{attribute addProperty BoxType "IODEVICETYPE_ETHERCATPROT"}
{attribute addProperty Id "DevCtrlAT %Q*UINT1620Frm0CtrlAT %Q*UINT1620Frm0WcCtrlAT %Q*UINT1620Frm1CtrlAT %Q*UINT1620Frm1WcCtrlAT %Q*UINT1620Frm2CtrlAT %Q*UINT1620Frm2WcCtrlAT %Q*UINT1620Frm3CtrlAT %Q*UINT1620Frm3WcCtrlAT %Q*UINT1620Frm4CtrlAT %Q*UINT1620Frm4WcCtrlAT %Q*UINT1620Frm5CtrlAT %Q*UINT1620Frm5WcCtrlAT %Q*UINT1620Frm6CtrlAT %Q*UINT1620Frm6WcCtrlAT %Q*UINT1620Frm7CtrlAT %Q*UINT1620Frm7WcCtrlAT %Q*UINT1620Frm8CtrlAT %Q*UINT1620Frm8WcCtrlAT %Q*UINT1620Frm9CtrlAT %Q*UINT1620Frm9WcCtrlAT %Q*UINT1620Frm10CtrlAT %Q*UINT1620Frm10WcCtrlAT %Q*UINT1620Frm11CtrlAT %Q*UINT1620Frm11WcCtrlAT %Q*UINT1620Frm12CtrlAT %Q*UINT1620Frm12WcCtrlAT %Q*UINT1620Frm13CtrlAT %Q*UINT1620Frm13WcCtrlAT %Q*UINT1620Frm14CtrlAT %Q*UINT1620Frm14WcCtrlAT %Q*UINT1620Frm15CtrlAT %Q*UINT1620Frm15WcCtrlAT %Q*UINT1620Frm16CtrlAT %Q*UINT1620Frm16WcCtrlAT %Q*UINT1620Frm17CtrlAT %Q*UINT1620Frm17WcCtrlAT %Q*UINT1620Frm18CtrlAT %Q*UINT1620Frm18WcCtrlAT %Q*UINT1620Frm19CtrlAT %Q*UINT1620Frm19WcCtrlAT %Q*UINT1620Frm20CtrlAT %Q*UINT1620Frm20WcCtrlAT %Q*UINT1620Frm21CtrlAT %Q*UINT1620Frm21WcCtrlAT %Q*UINT1620Frm22CtrlAT %Q*UINT1620Frm22WcCtrlAT %Q*UINT1620Frm23CtrlAT %Q*UINT1620Frm23WcCtrlAT %Q*UINT1620Frm24CtrlAT %Q*UINT1620Frm24WcCtrlAT %Q*UINT1620Frm25CtrlAT %Q*UINT1620Frm25WcCtrlAT %Q*UINT1620"}
{attribute addProperty CRC "1204938755"}
{attribute addProperty SizeInBites "848"}
{attribute addProperty SizeInBytes "106"}
TYPE Outputs_47D1E803 :
STRUCT
	{attribute addProperty Name "DevCtrl"}
	DevCtrl AT %Q* : UINT;
	{attribute addProperty Name "Frm0Ctrl"}
	Frm0Ctrl AT %Q* : UINT;
	{attribute addProperty Name "Frm0WcCtrl"}
	Frm0WcCtrl AT %Q* : UINT;
	{attribute addProperty Name "Frm1Ctrl"}
	Frm1Ctrl AT %Q* : UINT;
	{attribute addProperty Name "Frm1WcCtrl"}
	Frm1WcCtrl AT %Q* : UINT;
	{attribute addProperty Name "Frm2Ctrl"}
	Frm2Ctrl AT %Q* : UINT;
	{attribute addProperty Name "Frm2WcCtrl"}
	Frm2WcCtrl AT %Q* : UINT;
	{attribute addProperty Name "Frm3Ctrl"}
	Frm3Ctrl AT %Q* : UINT;
	{attribute addProperty Name "Frm3WcCtrl"}
	Frm3WcCtrl AT %Q* : UINT;
	{attribute addProperty Name "Frm4Ctrl"}
	Frm4Ctrl AT %Q* : UINT;
	{attribute addProperty Name "Frm4WcCtrl"}
	Frm4WcCtrl AT %Q* : UINT;
	{attribute addProperty Name "Frm5Ctrl"}
	Frm5Ctrl AT %Q* : UINT;
	{attribute addProperty Name "Frm5WcCtrl"}
	Frm5WcCtrl AT %Q* : UINT;
	{attribute addProperty Name "Frm6Ctrl"}
	Frm6Ctrl AT %Q* : UINT;
	{attribute addProperty Name "Frm6WcCtrl"}
	Frm6WcCtrl AT %Q* : UINT;
	{attribute addProperty Name "Frm7Ctrl"}
	Frm7Ctrl AT %Q* : UINT;
	{attribute addProperty Name "Frm7WcCtrl"}
	Frm7WcCtrl AT %Q* : UINT;
	{attribute addProperty Name "Frm8Ctrl"}
	Frm8Ctrl AT %Q* : UINT;
	{attribute addProperty Name "Frm8WcCtrl"}
	Frm8WcCtrl AT %Q* : UINT;
	{attribute addProperty Name "Frm9Ctrl"}
	Frm9Ctrl AT %Q* : UINT;
	{attribute addProperty Name "Frm9WcCtrl"}
	Frm9WcCtrl AT %Q* : UINT;
	{attribute addProperty Name "Frm10Ctrl"}
	Frm10Ctrl AT %Q* : UINT;
	{attribute addProperty Name "Frm10WcCtrl"}
	Frm10WcCtrl AT %Q* : UINT;
	{attribute addProperty Name "Frm11Ctrl"}
	Frm11Ctrl AT %Q* : UINT;
	{attribute addProperty Name "Frm11WcCtrl"}
	Frm11WcCtrl AT %Q* : UINT;
	{attribute addProperty Name "Frm12Ctrl"}
	Frm12Ctrl AT %Q* : UINT;
	{attribute addProperty Name "Frm12WcCtrl"}
	Frm12WcCtrl AT %Q* : UINT;
	{attribute addProperty Name "Frm13Ctrl"}
	Frm13Ctrl AT %Q* : UINT;
	{attribute addProperty Name "Frm13WcCtrl"}
	Frm13WcCtrl AT %Q* : UINT;
	{attribute addProperty Name "Frm14Ctrl"}
	Frm14Ctrl AT %Q* : UINT;
	{attribute addProperty Name "Frm14WcCtrl"}
	Frm14WcCtrl AT %Q* : UINT;
	{attribute addProperty Name "Frm15Ctrl"}
	Frm15Ctrl AT %Q* : UINT;
	{attribute addProperty Name "Frm15WcCtrl"}
	Frm15WcCtrl AT %Q* : UINT;
	{attribute addProperty Name "Frm16Ctrl"}
	Frm16Ctrl AT %Q* : UINT;
	{attribute addProperty Name "Frm16WcCtrl"}
	Frm16WcCtrl AT %Q* : UINT;
	{attribute addProperty Name "Frm17Ctrl"}
	Frm17Ctrl AT %Q* : UINT;
	{attribute addProperty Name "Frm17WcCtrl"}
	Frm17WcCtrl AT %Q* : UINT;
	{attribute addProperty Name "Frm18Ctrl"}
	Frm18Ctrl AT %Q* : UINT;
	{attribute addProperty Name "Frm18WcCtrl"}
	Frm18WcCtrl AT %Q* : UINT;
	{attribute addProperty Name "Frm19Ctrl"}
	Frm19Ctrl AT %Q* : UINT;
	{attribute addProperty Name "Frm19WcCtrl"}
	Frm19WcCtrl AT %Q* : UINT;
	{attribute addProperty Name "Frm20Ctrl"}
	Frm20Ctrl AT %Q* : UINT;
	{attribute addProperty Name "Frm20WcCtrl"}
	Frm20WcCtrl AT %Q* : UINT;
	{attribute addProperty Name "Frm21Ctrl"}
	Frm21Ctrl AT %Q* : UINT;
	{attribute addProperty Name "Frm21WcCtrl"}
	Frm21WcCtrl AT %Q* : UINT;
	{attribute addProperty Name "Frm22Ctrl"}
	Frm22Ctrl AT %Q* : UINT;
	{attribute addProperty Name "Frm22WcCtrl"}
	Frm22WcCtrl AT %Q* : UINT;
	{attribute addProperty Name "Frm23Ctrl"}
	Frm23Ctrl AT %Q* : UINT;
	{attribute addProperty Name "Frm23WcCtrl"}
	Frm23WcCtrl AT %Q* : UINT;
	{attribute addProperty Name "Frm24Ctrl"}
	Frm24Ctrl AT %Q* : UINT;
	{attribute addProperty Name "Frm24WcCtrl"}
	Frm24WcCtrl AT %Q* : UINT;
	{attribute addProperty Name "Frm25Ctrl"}
	Frm25Ctrl AT %Q* : UINT;
	{attribute addProperty Name "Frm25WcCtrl"}
	Frm25WcCtrl AT %Q* : UINT;
END_STRUCT
END_TYPE

(* stored: Version 1.2.0.0, ProductVersion 3.1.4024.9
   DUT Outputs_47D1E803: Id {dc65a96c-6b4b-443d-b9e2-f7bf2adb348f} *)
